// Block: Loop1_PERS

DATA_BLOCK Loop1_PERS
VERSION : 0.1
   NON_RETAIN
   VAR
      PersistentValues : Struct
         Par : SmartLoopControl_Par;
      END_STRUCT;
      AuxPE_LsMax_TP_Entry : Bool;
      AuxPE_LsMax_TP_Exit : Bool;
   END_VAR

BEGIN
   // No initialization required
END_DATA_BLOCK
